FUNCTION_BLOCK PUBLIC FB_CNC EXTENDS FB_EventLogger
VAR_INPUT
	CalibrationCam						: ARRAY[0..HLI_SYS_AX_MAXIDX] OF BOOL;
	LogAxisNo							: ARRAY[0..HLI_SYS_AX_MAXIDX] OF INT;// EtherCAT ID of Axis
	MaxChannelIdx						: INT := 0;	//Max index of channel that is used starting at 0, example: 1 -> totally 2 channels, maximum of 11 (12 channels) is allowed here *)
	Energize							: BOOL;// CNC Energised Flag
END_VAR
VAR_OUTPUT
	
END_VAR
VAR_IN_OUT	                			
	Control								: ST_System;
	Spindle								: ST_Spindle;						//Spindle interface	
END_VAR    
VAR 
	_AxisTorqueLimit					AT %Q* : ARRAY [0..4] OF UINT;								//Bipolar Torque Limit for axes (mapped from drive)
	_DrivePowerManagementStatusWords AT %I* :ARRAY [0..4] OF INT;									//Power management status to detect drives dropping power to ensure rehoming occurs.
	
	_Axis								: ARRAY[0..HLI_SYS_AX_MAXIDX] OF FB_CNCAxis;	//Axis data struct
	{attribute 'tc_no_symbol'}
	_Channel							: ARRAY[0..3] OF HLI3_CNCChannel;	//Channel data struct
	_MachineMode						: ARRAY[0..3] OF ST_MachineMode;	//Machine mode data struct
	_ManualMode							: ST_Selection;						//Manual Mode Selection
	_AutomaticMode						: ST_Selection;						//Automatic Mode Selection
	_MDIMode							: ST_Selection;						//MDI Mode Selection
	_HandwheelMode						: ST_Selection;						//Handwheel Mode Selection
	_StandbyMode						: ST_Selection;						//Standby Mode Selection
	_ReferenceMode						: ST_Selection;						//Reference Mode Selection
	_ManHome							: ST_Selection;						//Manual Home Selection
	_RetractTool						: ST_Selection;						//Retract tool from workpiece
	_SpindleWarmup						: ST_Selection;						//Warm up Spindle
	_AxisNames							: ARRAY[0..4] OF STRING;			//Individual Axis Names for HMI
	_AxisInManual						: ARRAY[0..4] OF BOOL;				//Axis in Manual Flag
	_SelectedChannel					: INT := 0;
	_SelectedAxis						: INT := 0;							//Axis Index Selected from HMI
	_SpindleVelocity					: UINT;								//Spindle Velocity Status
	_SpindleRev							: DINT;								//Spindle Revolution Command
	_AutoEn								: BOOL;								//Auto Enable
	_AutoHome							: BOOL;								//Command Home Drive Auto
	_AxisEnabled						: BOOL;								//All Axes are enabled
	_ManualModeJog						: BOOL;								//Manual Jog Mode
	_ManualModeInc						: BOOL;								//Manual Increment Mode
	_FeedOverride						: UINT := 100;
	_Fault								: BOOL;	     						//Device Fault
	_FaultTimer_ET						: REAL;								//Fault timer elapsed
	_Alarm								: BOOL;								//Device Alarm         
	_Warning							: BOOL;								//Device Warning   
	{attribute 'tc_no_symbol'}
	_ParkMDIString						: STRING;							//Parking MDI String   
	{attribute 'tc_no_symbol'}  
	_AlarmNum							: UDINT;							//Device Alarm Number  
	{attribute 'tc_no_symbol'}
	_WarningNum							: DINT;								//Device Warning Number
	{attribute 'tc_no_symbol'}
	_R_Trig								: ARRAY[0..19] OF R_TRIG;			//Private Rising Edge Triggers
	_HandwheelAxisIsSelected			: BOOL;								//True when axis selected on handwheel
	_Handwheel 							: ST_Handwheel; 					//Handwheel controller inputs
	_ProgramEnd							: ARRAY[0..3] OF BOOL;				//Program End
	_CurrentLine						: DINT;								//N function of currently running program (i.e. N60 -> 60)
	_CurrentNCProgram					: STRING;							//Program currently running in CNC kernal
	_NCProgramCode						: STRING(15000);					//Code of program for reloading into HMI text display\
END_VAR
VAR PERSISTENT                      	
	_Name								: STRING[15];						//Name for HMI
	_Description						: STRING[40];						//Description for HMI
	_AlarmMute							: BOOL;								//Alarm Mute
	_FaultTimer_PT						: REAL;								//Fault timer preset time	
	_Homed								: BOOL;								//Servo is Homed
	_Variables							: ARRAY [0..9] OF ST_Variable;				//Device Associated Varibles Array	
	_ToolData							: ARRAY [0..6] OF ST_CNC_TOOL_DATA_EXT;		//Data for tools
	_PositionOffset						: ARRAY[0..HLI_SYS_AX_MAXIDX] OF LREAL;		//Home position offsets for Axes
	_ParkPositions						: ARRAY[0..HLI_SYS_AX_MAXIDX] OF INT;		//Park positions for Axes
	_pVE_Chan0							: POINTER TO ST_VE_CHAN0;					//Channel 0 User defined Variables
	_Referencing						: E_CNC_HomingMethod; 						//Method to home
	_MeasurementOrder					: ARRAY[0..5] OF UINT :=[2,3,4,1,0];		//Measurement Axis Index Order i.e [2,3,4,1,0] Would be the same as G74 X5 Y4 Z1 C3 A2
	_MeasurementMDIString				: ARRAY[0..5] OF STRING := ['G100 X-10000$R$NM50$R$NM53$R$NG4 1$R$NM51$R$N#PUT AX [X] $R$NM52$R$N#CALL AX [X,11,0]$R$NM54$R$N',
																	'G100 Y-10000$R$NM50$R$NM53$R$NG4 1$R$NM51$R$N#PUT AX [Y] $R$NM52$R$N#CALL AX [Y,10,1]$R$NM54$R$N',
																	'G100 Z1000$R$NM50$R$NM53$R$NG4 1$R$NM51$R$N#PUT AX [Z] $R$NM52$R$N#CALL AX [Z,7,2]$R$NM54$R$N',
																	'G100 C-1000$R$NM50$R$NM53$R$NG4 1$R$NM51$R$N#PUT AX [C] $R$NM52$R$N#CALL AX [C,8,3]$R$NM54$R$N',
																	'G100 A1000$R$NM50$R$NM53$R$NG4 1$R$NM51$R$N#PUT AX [A] $R$NM52$R$N#CALL AX [A,9,4]$R$NM54$R$N',
																	''];//Measurement MDI String

END_VAR

HLI3_Init(); 
M_WarningMonitor();
M_AlarmMonitor();

(* Call CNC related code only if the HLI has been initialized succesfully! *)
IF CNCSystem.bHLIInit THEN
	M_AxesHandler();    	
	M_ManualMode(_Chan:= _SelectedChannel);
	M_ChannelHandler();	
	M_VariableViewer();	
	M_Selections(_Chan:= _SelectedChannel);	
	M_Spindle(_Chan:= _SelectedChannel);
	M_ToolHandler(_Chan:= _SelectedChannel);
	M_Homing(_Chan:= _SelectedChannel);

  //Mod from Local
  //Mod on local pre pull
END_IF

{attribute 'monitoring' := 'variable'}
PROPERTY PUBLIC Alarm : Bool
GET
Alarm := _Alarm;
END_GET
END_PROPERTY

{attribute 'monitoring' := 'variable'}
PROPERTY PUBLIC AlarmMute : BOOL
SET
AlarmMute := _AlarmMute;
END_SET
END_PROPERTY

{attribute 'monitoring' := 'variable'}
PROPERTY PUBLIC AutoHome : Bool
SET
_AutoHome := AutoHome;
END_SET
END_PROPERTY

{attribute 'monitoring' := 'variable'}
PROPERTY PUBLIC AxisEnabled : Bool
GET
AxisEnabled := _AxisEnabled;
END_GET
END_PROPERTY

{attribute 'monitoring' := 'variable'}
PROPERTY PUBLIC Description : String[40]
GET
Description := _Description;
END_GET
SET
_Description := Description;
END_SET
END_PROPERTY

{attribute 'monitoring' := 'variable'}
PROPERTY PUBLIC Fault : Bool
SET
_Fault := Fault;
END_SET
END_PROPERTY

{attribute 'monitoring' := 'variable'}
PROPERTY PUBLIC FaultTimer_ET : real
GET
FaultTimer_ET := _FaultTimer_ET;
END_GET
END_PROPERTY

{attribute 'monitoring' := 'variable'}
PROPERTY PUBLIC FaultTimer_PT : real
GET
FaultTimer_PT := _FaultTimer_PT;
END_GET
SET
_FaultTimer_PT := FaultTimer_PT;
END_SET
END_PROPERTY

PROPERTY PUBLIC FeedOverride : UINT
GET
FeedOverride:= _FeedOverride;
END_GET
SET
_FeedOverride:= FeedOverride;
END_SET
END_PROPERTY

PROPERTY PUBLIC HandwheelSelected : BOOL
GET
HandwheelSelected:= (_MachineMode[0].ManualMode.nManualTyp = 1);
END_GET
END_PROPERTY

{attribute 'monitoring' := 'variable'}
PROPERTY PUBLIC Homed : Bool
GET
Homed := _Homed;
END_GET
END_PROPERTY

METHOD PRIVATE M_AlarmMonitor
VAR_INPUT
END_VAR
VAR_INST // added by the converter: edge detectors and wires of the graphical bodies
    _w1, _w2, _w3, _w4, _w5 : BOOL;
    _rt1 : R_TRIG;
END_VAR
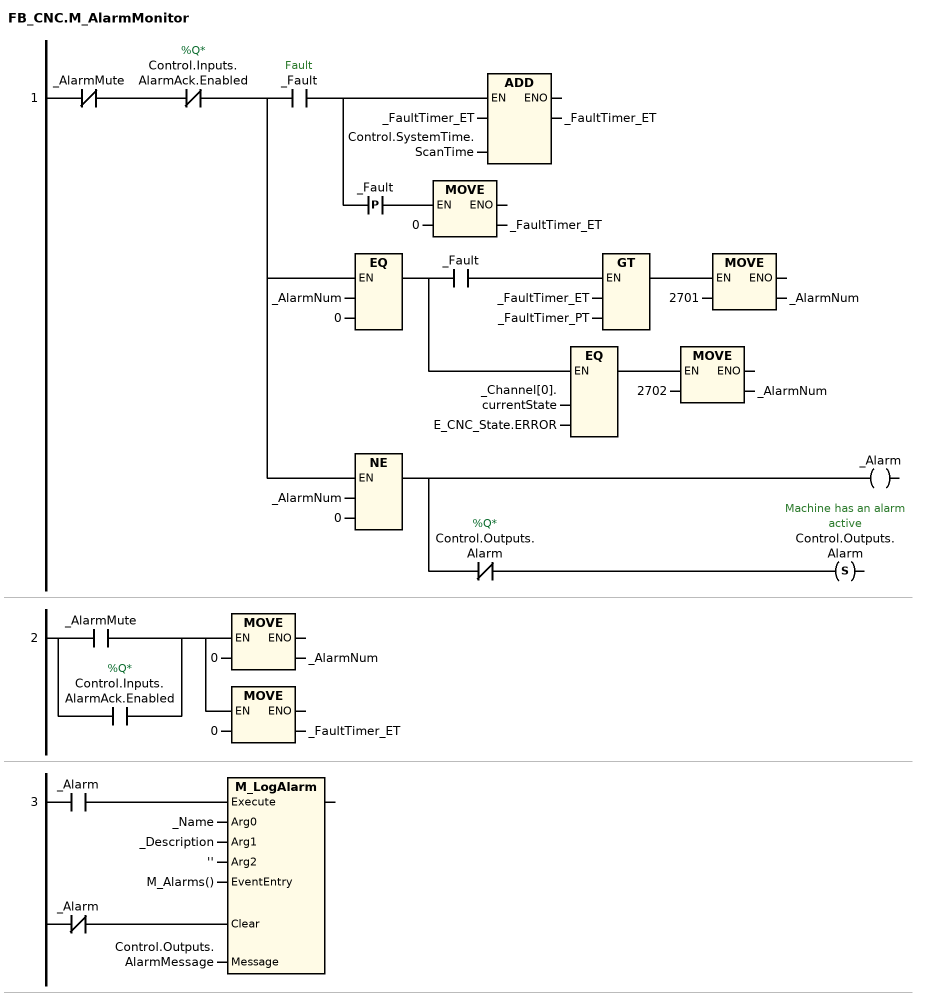
// NETWORK 1
//   Control.Inputs.AlarmAck.Enabled: AT %Q*
//   _Fault: Fault
//   _FaultTimer_ET: Fault timer elapsed
//   Control.SystemTime.ScanTime: Last scan time (Seconds)
//   _FaultTimer_PT: Fault timer preset time
//   Control.Outputs.Alarm: AT %Q* | Machine has an alarm active
_w1 := NOT _AlarmMute AND NOT Control.Inputs.AlarmAck.Enabled;
_w2 := _w1 AND _Fault;
IF _w2 THEN _FaultTimer_ET := _FaultTimer_ET + Control.SystemTime.ScanTime; END_IF
_rt1(CLK := _Fault);
IF _w2 AND _rt1.Q THEN _FaultTimer_ET := 0; END_IF
_w3 := _w1 AND _AlarmNum = 0;
IF _w3 AND _Fault AND _FaultTimer_ET > _FaultTimer_PT THEN _AlarmNum := 2701; END_IF
IF _w3 AND _Channel[0].currentState = E_CNC_State.ERROR THEN _AlarmNum := 2702; END_IF
_w4 := _w1 AND _AlarmNum <> 0;
_Alarm := _w4;
Control.Outputs.Alarm S= _w4 AND NOT Control.Outputs.Alarm;

// NETWORK 2
//   Control.Inputs.AlarmAck.Enabled: AT %Q*
//   _FaultTimer_ET: Fault timer elapsed
_w5 := _AlarmMute OR Control.Inputs.AlarmAck.Enabled;
IF _w5 THEN _AlarmNum := 0; END_IF
IF _w5 THEN _FaultTimer_ET := 0; END_IF

// NETWORK 3
M_LogAlarm(Execute := _Alarm, Arg0 := _Name, Arg1 := _Description, Arg2 := '', EventEntry := M_Alarms(), Clear := NOT _Alarm, Message := Control.Outputs.AlarmMessage);
END_METHOD

METHOD PRIVATE M_Alarms : TcEventEntry
VAR_INPUT
END_VAR
CASE _AlarmNum OF
	2701: M_Alarms:= TC_Events.TcCnc.A_2701;//Alarm	
	2702: M_Alarms:= TC_Events.TcCnc.A_2702;//Mode Error					
ELSE
	M_Alarms:= TC_Events.TcCnc.A_Undefined;
END_CASE
END_METHOD

METHOD PRIVATE M_AxesHandler
VAR_INST
	{attribute 'tc_no_symbol'}
	_HliAxisIdx					: INT;				//Loop index	
	{attribute 'tc_no_symbol'}			
	_FirstSpindle				: INT := -1;		//Spindle HLI index
	{attribute 'tc_no_symbol'}
	_fbAxesError 				: FB_AxesError;		//Axes error
END_VAR
_fbAxesError(bReset := (_Alarm AND Control.Inputs.AlarmAck.Enabled));
_AxisEnabled := TRUE;   
FOR _HliAxisIdx := 0 TO UDINT_TO_INT(gNrAx-1) DO			
	_Axis[_HliAxisIdx](bCalibrationCam:= CalibrationCam[_HliAxisIdx],
		bEnable	:= _AutoEn,
		nLogAxisNo := LogAxisNo[_HliAxisIdx]);
	_Axis[_HliAxisIdx].stOptions.bProbingSignal:= CalibrationCam[_HliAxisIdx];
		
	IF _HliAxisIdx <= UDINT_TO_INT(gNrAx-2) THEN
		_AxisNames[_HliAxisIdx] := gpCh[0]^.bahn_state.coord_r[_HliAxisIdx].axis_name_r.zeichen;
		_AxisInManual[_HliAxisIdx] := _MachineMode[0].ManualMode.nLogAxisNumber = INT_TO_UINT(_Axis[_HliAxisIdx].nLogAxisNo);
		_Axis[_HliAxisIdx].stOptions.bProbingSignal := CalibrationCam[_HliAxisIdx];	
		IF (NOT _Axis[_HliAxisIdx].stStatus.bIsEnabled) THEN    // if one axis status is "not enabled" -> reset PLCStatusAxisEnabled
			_AxisEnabled := FALSE;
		END_IF
	END_IF
		
		IF HLI3_CheckAxisValid(_HliAxisIdx) THEN
			IF _FirstSpindle = -1 AND gpAx[_HliAxisIdx]^.ipo_state.spindle_axis_r THEN  (* store HLIIndex of first spindle *)
				_FirstSpindle := _HliAxisIdx;
			END_IF
		END_IF
		
END_FOR
END_METHOD

METHOD M_ChannelHandler
VAR_INST
	{attribute 'tc_no_symbol'}
	_Chan					: INT;								//Channel index
	{attribute 'tc_no_symbol'}
	_OldSelectedChannel		: UDINT;							//Previous channel index
	{attribute 'tc_no_symbol'}
	_stOptions				: ST_CNC_CH_Options;				//HLI options for structure 
	{attribute 'tc_no_symbol'}
	_ChannelSignals			: ST_ChannelSignals;				//HLI channel signal structure
	{attribute 'tc_no_symbol'}
	_BlockSearch			: ARRAY[0..3] OF HLI3_BlockSearch;	//HLI block search structure
	{attribute 'tc_no_symbol'}
	_ErrorHandler			: ARRAY[0..3] OF FB_ChannelError;	//HLI channel error structure				
END_VAR
IF (_OldSelectedChannel <>INT_TO_UDINT(_SelectedChannel)) THEN
	_ChannelSignals.SingleBlock 		:= _MachineMode[_SelectedChannel].ChannelSignals.SingleBlock;
	_ChannelSignals.PrgBlockIgnore		:= _MachineMode[_SelectedChannel].ChannelSignals.PrgBlockIgnore;
	_ChannelSignals.M01Stop 			:= _MachineMode[_SelectedChannel].ChannelSignals.M01Stop;
	_ChannelSignals.Backward 			:= _MachineMode[_SelectedChannel].ChannelSignals.Backward;
	_ChannelSignals.FeedHold 			:= _MachineMode[_SelectedChannel].ChannelSignals.FeedHold;
	_OldSelectedChannel 				:= INT_TO_UDINT(_SelectedChannel);
END_IF

_MachineMode[_SelectedChannel].ChannelSignals.SingleBlock 	:= _ChannelSignals.SingleBlock;
_MachineMode[_SelectedChannel].ChannelSignals.PrgBlockIgnore:= _ChannelSignals.PrgBlockIgnore;
_MachineMode[_SelectedChannel].ChannelSignals.M01Stop 		:= _ChannelSignals.M01Stop;
_MachineMode[_SelectedChannel].ChannelSignals.Backward 		:= _ChannelSignals.Backward;
_MachineMode[_SelectedChannel].ChannelSignals.FeedHold 		:= _ChannelSignals.FeedHold;

_stOptions.bReferenceModeStartRequired := FALSE;
//_stOptions.bDisableCNCPLCWatchDog := TRUE;

FOR _Chan := 0 TO MaxChannelIdx DO
	IF (HLI3_CheckChannelValid(_Chan)) THEN		
		
		_MachineMode[_Chan].Mode 	:= _Channel[_Chan].currentMode;
		_MachineMode[_Chan].State	:= _Channel[_Chan].currentState;
		_ErrorHandler[_Chan](nChanIdx	:= _Chan);				

		_Channel[_Chan]
			(nChanIdx			:= _Chan,							
			 bModeStandby		:= _MachineMode[_Chan].Standby,
			 bModeAutomatic		:= _MachineMode[_Chan].Automatic,
			 bModeManual		:= _MachineMode[_Chan].Manual,
			 bModeMDI			:= _MachineMode[_Chan].MDI,	 
			 bModeReference		:= _MachineMode[_Chan].Homing,
			 bStateSelect		:= _MachineMode[_Chan].Select,
			 bStateReady		:= _MachineMode[_Chan].Ready,
			 bStateStart		:= _MachineMode[_Chan].Start,
			 bStateStop			:= _MachineMode[_Chan].Stop,
			 bStateReset		:= _MachineMode[_Chan].Reset,
			 nFeedOverride		:= _FeedOverride * 10,
			 nRapidFeedOverride := _FeedOverride * 10, 
			 sProgramName		:= _MachineMode[_Chan].ProgramName,			 
			 sMDIString			:= _MachineMode[_Chan].MDIString,
			 bBackwardMotion	:= _MachineMode[_Chan].ChannelSignals.Backward,
			 bPrgBlockIgnore	:= _MachineMode[_Chan].ChannelSignals.PrgBlockIgnore,
			 bFeedHold			:= _MachineMode[_Chan].ChannelSignals.FeedHold,
			 bSingleBlock		:= _MachineMode[_Chan].ChannelSignals.SingleBlock,
			 bDoSingleBlock		:= _MachineMode[_Chan].ChannelSignals.DoSingleBlock,
			 bM01Stop			:= _MachineMode[_Chan].ChannelSignals.M01Stop,
			 nSyntaxCheck		:= _MachineMode[_Chan].SyntaxCheck.nType,
			 bM30Acknowledgement:= TRUE,
			 stManualModeParameter  	 	 := stManualModeParameter[_Chan],
			 stManualModeControlElements	 := stManualModeControlElements[_Chan],
			 stManualModeControlElementState := stManualModeControlElementState,
			 stOptions			:= 	_stOptions
			);
			
		_r_trig[_Chan](CLK:= gpCh[_Chan]^.bahn_state.program_end_r);
		_ProgramEnd[_Chan]:= _r_trig[_Chan].Q;
		
		_BlockSearch[_Chan]
			(nChanIdx			:= _Chan,
			 bStartRead      	:= _MachineMode[_Chan].BlockSearch.bStartRead,   (* Edge signal *)
			 bStartWrite     	:= _MachineMode[_Chan].BlockSearch.bStartWrite,  (* Edge signal *)
			 BlockSearch		:= _MachineMode[_Chan].BlockSearch
			);
		
		CNCSystem.Channel[_Chan].ActDistance 	:= DINT_TO_LREAL(_BlockSearch[_Chan].coveredDistance_AfterReset) / 10.0;
		CNCSystem.Channel[_Chan].ActBlockCount 	:= _BlockSearch[_Chan].actualBlockCount_AfterReset;
						
	END_IF
END_FOR

_CurrentNCProgram := gpCh[0]^.bahn_state.file_name_r.zeichen;
_CurrentLine:= gpCh[0]^.bahn_state.block_nr_r;
END_METHOD

METHOD PRIVATE M_Homing
VAR_INPUT
	{attribute 'tc_no_symbol'}
	_Chan								 : INT;									//Channel index
END_VAR
VAR_INST
	{attribute 'tc_no_symbol'}
	_Step                  			 	 : ARRAY[0..3] OF INT;					//Step counter
	{attribute 'tc_no_symbol'}
	_Axe					 			 : UINT;								//Axes index
	{attribute 'tc_no_symbol'}
	_SetDrivePosition					 : BOOL;								//Set drive position
	{attribute 'tc_no_symbol'}
	_DeleteDrivePosition				 : BOOL;								//Delete drive position
	{attribute 'tc_no_symbol'}	
	_fb_CNCAX5000SetPositionOffset		 : FB_CNCAX5000SetPositionOffset;		//Sets encoder position in drive memory
	{attribute 'tc_no_symbol'}
	_fb_CNCAX5000DeletePositionOffset	 : FB_CNCAX5000DeletePositionOffset;	//Clears drive memory
END_VAR
IF _MachineMode[_Chan].State = E_CNC_State.ERROR OR Control.PackMLState.Stopped THEN
   _Step[_Chan] := 0;
END_IF
 
CASE _Referencing OF

//Homing Method with Calibration Cam. This method uses the Position Offsets stored in the CNC Params. The encoder position is NOT stored in memory.
E_CNC_HomingMethod.Homing:

	CASE _Step[_Chan] OF
		0: //Idle
			IF _AutoHome AND NOT _Alarm THEN
				_Homed := FALSE;
				_Axe:=0;
			    _Step[_Chan] := 1;
			ELSIF _ManHome.Queued AND NOT _Alarm THEN
				_Homed := FALSE;
				IF _ManHome.Enabled THEN
					_Axe:=INT_TO_UINT(_SelectedAxis);
					_Step[_Chan] := 10;
				END_IF
			END_IF
		
		1://Update Homing Offsets
			_Axis[0].fRefOffset:= _PositionOffset[0];
			_Axis[0].bSetRefOffset:= TRUE;
			_Axis[1].fRefOffset:= _PositionOffset[1];
			_Axis[1].bSetRefOffset:= TRUE;
			_Axis[2].fRefOffset:= _PositionOffset[2];
			_Axis[2].bSetRefOffset:= TRUE;
			_Axis[3].fRefOffset:= _PositionOffset[3];
			_Axis[3].bSetRefOffset:= TRUE;
			_Axis[4].fRefOffset:= _PositionOffset[4];
			_Axis[4].bSetRefOffset:= TRUE;

			_Step[_Chan] := 2;
	
	
		2://Enable Homing
			_MachineMode[0].Homing:= TRUE;

			IF _Axis[0].stStatus.bHomingDone AND _Axis[1].stStatus.bHomingDone AND 
				_Axis[2].stStatus.bHomingDone AND _Axis[3].stStatus.bHomingDone AND _Axis[4].stStatus.bHomingDone THEN
					_Step[_Chan] := 3;
			END_IF
	
		3: //Wait for CNC to reach park positions
		 	IF _MachineMode[_Chan].State = E_CNC_State.READY THEN
		     	_Step[_Chan] := 4;
		 	END_IF
		
		4://Set mode to standby	
			_Homed := TRUE;
			_MachineMode[_Chan].Standby := TRUE;
			IF NOT _Autohome AND NOT _ManHome.Enabled AND _MachineMode[_Chan].Mode = E_CNC_Mode.STANDBY_MODE THEN
				_Step[_Chan] := 0;
			END_IF
			
		//Single Axis Manual Home
		10://Set MDI Mode
			_MachineMode[_Chan].MDI := TRUE;
			IF _MachineMode[_Chan].Mode = E_CNC_Mode.MDI_MODE THEN
				_Step[_Chan] := 11;
	    	END_IF
			
		11://Set homing string for indiviudal axis
			CASE _Axe OF
				0: _MachineMode[_Chan].MDIString := 'G74 X0';
				1: _MachineMode[_Chan].MDIString := 'G74 Y0';
				2: _MachineMode[_Chan].MDIString := 'G74 Z0';
				3: _MachineMode[_Chan].MDIString := 'G74 C0';
				4: _MachineMode[_Chan].MDIString := 'G74 A0';
			END_CASE
			_MachineMode[_Chan].Start := TRUE;
			_SetDrivePosition := FALSE;
	 		_Step[_Chan] := 12;
			
		12://Wait for CNC ready state
			IF _MachineMode[_Chan].State = E_CNC_State.READY THEN
	       		_Step[_Chan] := 13;
	    	END_IF
			
		13://Park Axis
			_MachineMode[_Chan].MDIString := CONCAT(_AxisNames[_SelectedAxis],TO_STRING(_ParkPositions[_SelectedAxis]));
			_MachineMode[_Chan].Start := TRUE;
			_Step[_Chan] := 14;
		
		14: //Wait for CNC to start moving to park positions
		 	IF _MachineMode[_Chan].State = E_CNC_State.ACTIVE THEN
		     	_Step[_Chan] := 15;
		 	END_IF		
			
		15: //Wait for CNC to reach park positions
		 	IF _MachineMode[_Chan].State = E_CNC_State.READY THEN
		     	_Step[_Chan] := 16;
		 	END_IF
		
		16://Set mode to standby	
			_Homed := TRUE;
			_MachineMode[_Chan].Standby := TRUE;
			IF NOT _Autohome AND NOT _ManHome.Enabled AND _MachineMode[_Chan].Mode = E_CNC_Mode.STANDBY_MODE THEN
				_Step[_Chan] := 0;
			END_IF
	END_CASE		


//Measurement Method With Probing Signal. This method uses the Position Offsets stored in the PLC. The encoder position IS stored in memory.
E_CNC_HomingMethod.Measurment:

	CASE _Step[_Chan] OF
		0: //Idle
			IF _AutoHome AND NOT _Alarm THEN
				_SetDrivePosition := FALSE;
				FOR _Axe := 0 TO UDINT_TO_UINT(gNrAx-2) DO
					_Axis[_MeasurementOrder[_Axe]].bSetRefOffset := FALSE;
					_Axis[_MeasurementOrder[_Axe]].stOptions.bResetCalibration := TRUE;
				END_FOR;
				_Homed := FALSE;
				_Axe:= 0;
			    _Step[_Chan] := 1;
			ELSIF _ManHome.Queued AND NOT _Alarm THEN
				_Homed := FALSE;
				IF _ManHome.Enabled THEN
					_Axe:=INT_TO_UINT(_SelectedAxis);
					_Step[_Chan] := 1;
				END_IF
			END_IF
			
		1://Enable Axes and set Standby Mode
			_AutoEn := TRUE;
			_MachineMode[_Chan].Standby := TRUE;
			IF _AxisEnabled AND _MachineMode[_Chan].Mode = E_CNC_Mode.STANDBY_MODE THEN
				_Step[_Chan] := 2;
			END_IF
	    	
	    2: //Set MDI mode
			_MachineMode[_Chan].MDI := TRUE;
			IF _MachineMode[_Chan].Mode = E_CNC_Mode.MDI_MODE THEN
				_Step[_Chan] := 3;
	    	END_IF
			
		3: //Reset homing done bool to allow ignorance of software limits
			IF _Axis[_MeasurementOrder[_Axe]].stStatus.bHomingDone = FALSE THEN
				_Axis[_MeasurementOrder[_Axe]].stOptions.bResetCalibration := FALSE;	
				_Step[_Chan] := 4;
			END_IF
			
	    4: //Create homing MDI string
			IF _ManHome.Enabled THEN
				_MachineMode[_Chan].MDIString := _MeasurementMDIString[_Axe];
			ELSE
				_MachineMode[_Chan].MDIString := _MeasurementMDIString[_MeasurementOrder[_Axe]];	
			END_IF
			_MachineMode[_Chan].Start := TRUE;
			_SetDrivePosition := FALSE;
	 		_Step[_Chan] := 5;
		
	    5: //Wait for CNC to start moving to home positions
	    	IF _MachineMode[_Chan].State = E_CNC_State.ACTIVE THEN
	       		_Step[_Chan] := 6;
	    	END_IF	
	
		6://Wait for CNC to reach home positions
		
				//M50 Clear Reference Flag
				IF CNCSystem.Channel[0].M[50].bState_rw THEN
					_Axis[_MeasurementOrder[_Axe]].stOptions.bResetCalibration := TRUE;
					IF _Axis[_MeasurementOrder[_Axe]].stStatus.bHomingDone = FALSE THEN
						_Axis[_MeasurementOrder[_Axe]].stOptions.bResetCalibration := FALSE;
						CNCSystem.Channel[0].M[50].bState_rw := FALSE;
					END_IF
				END_IF
				
				//M51 Set Drive Position
				IF CNCSystem.Channel[0].M[51].bState_rw THEN
					_SetDrivePosition := TRUE;
				END_IF
				IF _Axis[_MeasurementOrder[_Axe]].stStatus.fActPosACS > (_PositionOffset[_MeasurementOrder[_Axe]] -1) AND  _Axis[_MeasurementOrder[_Axe]].stStatus.fActPosACS < (_PositionOffset[_MeasurementOrder[_Axe]] +1) THEN
					CNCSystem.Channel[0].M[51].bState_rw := FALSE;
					_SetDrivePosition := FALSE;
				END_IF 
				
				//M52 Set Axis as Homed
				IF CNCSystem.Channel[0].M[52].bState_rw THEN
					_Axis[_MeasurementOrder[_Axe]].fRefOffset := 0;
					_Axis[_MeasurementOrder[_Axe]].bSetRefOffset := TRUE;
					IF _Axis[_MeasurementOrder[_Axe]].stStatus.bHomingDone = TRUE THEN
						CNCSystem.Channel[0].M[52].bState_rw := FALSE;
						_Axis[_MeasurementOrder[_Axe]].bSetRefOffset := FALSE;
					END_IF
				END_IF
				
				//M53 Disable Axis
				IF CNCSystem.Channel[0].M[53].bState_rw THEN
					_AutoEn := FALSE;
					IF NOT _Axis[_MeasurementOrder[_Axe]].stStatus.bIsEnabled THEN
						CNCSystem.Channel[0].M[53].bState_rw := FALSE;
					END_IF
				END_IF
				
				//M54 Enable Axis
				IF CNCSystem.Channel[0].M[54].bState_rw THEN
					_AutoEn := TRUE;
					IF _Axis[_MeasurementOrder[_Axe]].stStatus.bIsEnabled THEN
						CNCSystem.Channel[0].M[54].bState_rw := FALSE;
						_Step[_Chan] := 7;	
					END_IF
				END_IF
				
	    7: //Wait for CNC to be Ready
	    	IF _MachineMode[_Chan].State = E_CNC_State.READY THEN
	       		IF (_ManHome.Enabled OR _Axe >= (gNrAx-3)) THEN//)>= 1 THEN
					_Step[_Chan] := 8;
				ELSE
					_Axe:=_Axe+1;
					_Step[_Chan] := 3;
				END_IF
	    	END_IF	
				
		8://Create parking MDI string
			IF _ManHome.Enabled THEN
				_ParkMDIString := CONCAT(_AxisNames[_SelectedAxis],TO_STRING(_ParkPositions[_SelectedAxis]));
			ELSE	
				FOR _Axe := 0 TO UDINT_TO_UINT(gNrAx-2) BY 1 DO	
					IF _Axe = 0 THEN
						_ParkMDIString	:= concat(_AxisNames[_Axe],TO_STRING(_ParkPositions[_Axe]));
					ELSE
						_ParkMDIString	:= concat(_ParkMDIString,concat(' ', concat(_AxisNames[_Axe],TO_STRING(_ParkPositions[_Axe]))));
					END_IF
				END_FOR	
			END_IF
			_MachineMode[_Chan].MDIString := _ParkMDIString;
			_MachineMode[_Chan].Start := TRUE;
			_Step[_Chan] := 9;
		
		9: //Wait for CNC to start moving to park positions
		 	IF _MachineMode[_Chan].State = E_CNC_State.ACTIVE THEN
		     	_Step[_Chan] := 10;
		 	END_IF		
			
		10: //Wait for CNC to reach park positions
		 	IF _MachineMode[_Chan].State = E_CNC_State.READY THEN
		     	_Step[_Chan] := 11;
		 	END_IF
		
		11://Set mode to standby	
			_Homed := TRUE;
			_MachineMode[_Chan].Standby := TRUE;
			IF NOT _Autohome AND NOT _ManHome.Enabled AND _MachineMode[_Chan].Mode = E_CNC_Mode.STANDBY_MODE THEN
				_Step[_Chan] := 0;
			END_IF
			
	END_CASE

END_CASE

//Delete Position Offset
_fb_CNCAX5000DeletePositionOffset(nLogAxisNo:= TO_UINT(_Axis[_MeasurementOrder[_Axe]].nLogAxisNo), Execute:= _DeleteDrivePosition, Memory:= tc3_cnc_drive.E_PositionOffsetMemory.ePositionOffsetMemory_Drive);

//Set Position Offset
_fb_CNCAX5000SetPositionOffset(nLogAxisNo:= TO_UINT(_Axis[_MeasurementOrder[_Axe]].nLogAxisNo), Execute:= _SetDrivePosition, Position:= _PositionOffset[_MeasurementOrder[_Axe]], Memory:= tc3_cnc_drive.E_PositionOffsetMemory.ePositionOffsetMemory_Drive);
END_METHOD

METHOD PRIVATE M_ManualMode
VAR_INPUT
	{attribute 'tc_no_symbol'}
	_Chan								 : INT;									//Channel index
END_VAR	
VAR_INST
	{attribute 'tc_no_symbol'}
	_fbUintUdInt						 : ARRAY [0..3] OF FB_Uint_Udint;		//Uint to udint FB
	{attribute 'tc_no_symbol'}
	_HandWheelBig						 : UDINT;								//Handwheel value
END_VAR
IF (HLI3_CheckChannelValid(_Chan)) THEN

	stManualModeParameter[_Chan].stChannelParameter.nChanIdx := _Chan;       (* Channel 1 *)
	stManualModeParameter[_Chan].stChannelParameter.nInc := _MachineMode[_Chan].ManualMode.nInc * 10;
	stManualModeParameter[_Chan].stChannelParameter.bG200ConfigurationViaPLC := TRUE;		
	
	stManualModeParameter[_Chan].stChannelParameter.eManualType := UINT_TO_INT(_MachineMode[_Chan].ManualMode.nManualTyp);			
	IF (stManualModeParameter[_Chan].stChannelParameter.eManualType = E_CNC_ManualType.Handwheel AND _Chan <> _SelectedChannel) THEN	(* if in Handwheel mode and the channel is NOT selected -> leave handwheel mode and change to TippMode*)
		stManualModeParameter[_Chan].stChannelParameter.eManualType := E_CNC_ManualType.TippMode;
	END_IF		
	
	stManualModeParameter[_Chan].stChannelParameter.stManualOption.bTrafoActive := _MachineMode[_Chan].ManualMode.stManualOption.bTrafoActive;
	stManualModeParameter[_Chan].stChannelParameter.stManualOption.bEcsActive := _MachineMode[_Chan].ManualMode.stManualOption.bEcsActive;
	stManualModeParameter[_Chan].stChannelParameter.stManualOption.eZeroOffset := _MachineMode[_Chan].ManualMode.stManualOption.eZeroOffset;					

	_ManualModeJog:=(_MachineMode[_SelectedChannel].ManualMode.nManualTyp=2) AND _Channel[_SelectedChannel].stCmdModesStates.stModes.Manual;
	_ManualModeInc:=(_MachineMode[_SelectedChannel].ManualMode.nManualTyp=3) AND _Channel[_SelectedChannel].stCmdModesStates.stModes.Manual;
	
	stManualModeParameter[_Chan].stAxisParameter.stControlUnit[0].nLogAxisNr := _MachineMode[_Chan].ManualMode.nLogAxisNumber;   (* Log. Achs Nummer *)
	IF stManualModeParameter[_Chan].stAxisParameter.stControlUnit[0].nLogAxisNr = 0 THEN
		stManualModeParameter[_Chan].stAxisParameter.stControlUnit[0].nLogAxisNr := gpCh[_Chan]^.bahn_state.coord_r[0].log_achs_nr_r;
		_MachineMode[_Chan].ManualMode.nLogAxisNumber := gpCh[_Chan]^.bahn_state.coord_r[0].log_achs_nr_r;
	END_IF
	stManualModeParameter[_Chan].stAxisParameter.stControlUnit[0].nSpeed := LREAL_TO_UDINT(_MachineMode[_Chan].ManualMode.nSpeed * (100000/60));//um/min >> mm/sec
	stManualModeControlElements[_Chan].stControlKeys[0].bKeyNeg := _MachineMode[_Chan].ManualMode.bKeyNeg;
	stManualModeControlElements[_Chan].stControlKeys[0].bKeyPos := _MachineMode[_Chan].ManualMode.bKeyPos;
	stManualModeControlElements[_Chan].stControlKeys[0].bKeyRapid := _MachineMode[_Chan].ManualMode.bKeyRapid;
	
	//Handwheel
	IF _Handwheel.xAxisSelect THEN
		_MachineMode[_Chan].ManualMode.nLogAxisNumber := INT_TO_UINT(_Axis[0].nLogAxisNo);
	ELSIF _Handwheel.yAxisSelect THEN
		_MachineMode[_Chan].ManualMode.nLogAxisNumber := INT_TO_UINT(_Axis[1].nLogAxisNo);
	ELSIF _Handwheel.zAxisSelect THEN
		_MachineMode[_Chan].ManualMode.nLogAxisNumber := INT_TO_UINT(_Axis[2].nLogAxisNo);
	ELSIF _Handwheel.aAxisSelect THEN
		_MachineMode[_Chan].ManualMode.nLogAxisNumber := INT_TO_UINT(_Axis[3].nLogAxisNo);
	ELSIF _Handwheel.cAxisSelect THEN
		_MachineMode[_Chan].ManualMode.nLogAxisNumber := INT_TO_UINT(_Axis[4].nLogAxisNo);
	ELSIF _MachineMode[_Chan].ManualMode.nManualTyp = 1 THEN
		_MachineMode[_Chan].ManualMode.nManualTyp := 0;			
	END_IF
	
	IF _Handwheel.x10Resolution THEN
		_MachineMode[_Chan].ManualMode.nHwResolution := 10;
	ELSIF _Handwheel.x100Resolution THEN
		_MachineMode[_Chan].ManualMode.nHwResolution := 100;
	ELSE
		_MachineMode[_Chan].ManualMode.nHwResolution := 1;
	END_IF
		
	stManualModeParameter[_Chan].stChannelParameter.nHandwheelResolution := UDINT_TO_DINT(_MachineMode[_Chan].ManualMode.nHwResolution)* LREAL_TO_DINT(10000);
	_fbUintUdint[_Chan](ninSmall := _Handwheel.Handwheel, nBig := _HandWheelBig);
	stManualModeControlElements[_Chan].nHandwheelinc[0] :=  UDINT_TO_DINT(_HandWheelBig);
	IF _HandWheelBig > 214748364 OR _HandWheelBig = 0 THEN
		_MachineMode[_Chan].ManualMode.nLogAxisNumber := 0;
		_HandWheelBig := 107374182;
	END_IF
END_IF
END_METHOD

METHOD PRIVATE M_Selections
VAR_INPUT
	{attribute 'tc_no_symbol'}
	_Chan					 : INT;
END_VAR
VAR_INST
END_VAR
//Reset
	_MachineMode[_Chan].Reset := Control.Inputs.AlarmAck.Enabled OR Control.Inputs.Reset.Enabled;

//Energize
	_R_Trig[7](CLK:=Energize); 
	IF _R_Trig[7].Q THEN 
		_AutoEn:= TRUE; 
	END_IF
	
	_R_trig[6](CLK:= NOT Energize); 
	IF _R_Trig[6].Q THEN 
		_AutoEn:= FALSE; 
	END_IF

//Stop
	_R_Trig[8](CLK:=Control.PackMLState.Stopping OR Control.PackMLState.Holding);
	_MachineMode[_SelectedChannel].Stop := _R_Trig[8].Q;

//Start
	_R_Trig[9](CLK:= (Control.PackMLState.Starting OR Control.PackMLState.Execute) AND _AxisEnabled);
	_MachineMode[_SelectedChannel].Start := _R_Trig[9].Q;
	
//Standby Mode
	_StandbyMode.Interlock := Control.PackMLState.Execute  OR (_StandbyMode.Enabled AND _MachineMode[_Chan].Mode <> E_CNC_Mode.STANDBY_MODE);
	IF _StandbyMode.Interlock THEN 
		_StandbyMode.Messages := 'CNC Machine Must not be Executing for Standby Mode'; 
	END_IF;
	
	_StandbyMode.Select := (_StandbyMode.Select) AND NOT _StandbyMode.Interlock;
	IF NOT _StandbyMode.Select AND NOT _StandbyMode.Interlock THEN 
		_StandbyMode.Messages := 'CNC Ready for Standby Mode'; 
	END_IF;
	
	_StandbyMode.Queued := _StandbyMode.Select;
	IF _StandbyMode.Queued AND NOT _StandbyMode.Enabled THEN 
		_StandbyMode.Messages := 'CNC Standby Mode Selection Queued'; 
	END_IF;
	
	_R_Trig[10](CLK:= _StandbyMode.Queued); 
	IF _R_Trig[10].Q THEN 
		_MachineMode[_Chan].Standby := TRUE;
	END_IF;
	
	_StandbyMode.Enabled := _StandbyMode.Queued AND _MachineMode[_Chan].Mode = E_CNC_Mode.STANDBY_MODE;
	IF _StandbyMode.Enabled THEN 
		_StandbyMode.Messages := 'CNC Standby Mode Enabled'; 
	END_IF;

//Automatic Mode Selection
	_AutomaticMode.Interlock := Control.PackMLState.Execute AND NOT _AutomaticMode.Enabled OR (_AutomaticMode.Enabled AND _MachineMode[_Chan].Mode <> E_CNC_Mode.AUTOMATIC_MODE);
	IF _AutomaticMode.Interlock THEN 
		_AutomaticMode.Messages := 'CNC Machine Must not be Executing for Automatic Mode Selection'; 
	END_IF;
	
	_AutomaticMode.Select := _AutomaticMode.Select AND NOT _AutomaticMode.Interlock;
	IF NOT _AutomaticMode.Select AND NOT _AutomaticMode.Interlock THEN
 		_AutomaticMode.Messages := 'CNC Ready for Automatic Mode'; 
	END_IF;
	
	_AutomaticMode.Queued := _AutomaticMode.Select;
	IF _AutomaticMode.Queued AND NOT _AutomaticMode.Enabled THEN 
		_AutomaticMode.Messages := 'CNC Automatic Mode Selection Queued'; 
	END_IF;
	
	_R_Trig[11](CLK:= _AutomaticMode.Queued);
	IF _R_Trig[11].Q THEN 
		_MachineMode[_Chan].Automatic := TRUE;
	END_IF;
	
	_AutomaticMode.Enabled := _AutomaticMode.Queued AND _MachineMode[_Chan].Mode = E_CNC_Mode.AUTOMATIC_MODE;
	IF _AutomaticMode.Enabled THEN 
		_AutomaticMode.Messages := 'CNC Automatic Mode Enabled'; 
	END_IF;

//3 MDI Mode Selection
	_MDIMode.Interlock := Control.PackMLState.Execute AND NOT _MDIMode.Enabled  OR (_MDIMode.Enabled AND _MachineMode[_Chan].Mode <> E_CNC_Mode.MDI_MODE);
	IF _MDIMode.Interlock THEN 
		_MDIMode.Messages := 'CNC Machine Must not be Executing for MDI Mode Selection'; 
	END_IF;
	
	_MDIMode.Select := _MDIMode.Select AND NOT _MDIMode.Interlock;
	IF NOT _MDIMode.Select AND NOT _MDIMode.Interlock THEN 
		_MDIMode.Messages := 'CNC Ready for MDI Mode'; 
	END_IF;
	
	_MDIMode.Queued := _MDIMode.Select;
	IF _MDIMode.Queued AND NOT _MDIMode.Enabled THEN 
		_MDIMode.Messages := 'CNC MDI Mode Selection Queued'; 
	END_IF;
	
	_R_Trig[12](CLK:= _MDIMode.Queued); 
	IF _R_Trig[12].Q THEN 
		_MachineMode[_Chan].MDI:= TRUE;
	END_IF;

	_MDIMode.Enabled := _MDIMode.Queued AND _MachineMode[_Chan].Mode = E_CNC_Mode.MDI_MODE;
	IF _MDIMode.Enabled THEN 
		_MDIMode.Messages := 'CNC MDI Mode Enabled'; 
	END_IF;

//Manual Mode Selection
	_ManualMode.Interlock := (NOT control.PackMLState.Stopped AND NOT control.PackMLState.Idle)OR (_ManualMode.Enabled AND ((_MachineMode[_Chan].Mode <> E_CNC_Mode.MANUAL_MODE)OR _R_Trig[15].Q));
	IF _ManualMode.Interlock THEN 
		_ManualMode.Messages := 'CNC Must be in a Stopped or Idle State for Manual Mode'; 
	END_IF;	_R_Trig[13](CLK:= _ManualMode.Queued);
	
	_ManualMode.Select := _ManualMode.Select AND NOT _ManualMode.Interlock;
	IF NOT _ManualMode.Select AND NOT _ManualMode.Interlock THEN 
		_ManualMode.Messages := 'CNC Ready for Manual Mode'; 
	END_IF;
	
	_ManualMode.Queued := _ManualMode.Select;
	IF _ManualMode.Queued AND NOT _ManualMode.Enabled THEN 
		_ManualMode.Messages := 'CNC Manual Mode Selection Queued'; 
	END_IF;

	IF _R_Trig[13].Q THEN 
		_MachineMode[_Chan].ManualMode.nManualTyp := 2;  _MachineMode[_Chan].Manual := TRUE; 
	END_IF;
	
	_ManualMode.Enabled := _ManualMode.Queued AND (_MachineMode[_Chan].ManualMode.nManualTyp<>1) AND _MachineMode[_Chan].Mode = E_CNC_Mode.MANUAL_MODE;
	IF _ManualMode.Enabled THEN 
		_ManualMode.Messages := 'CNC Manual Mode Enabled';
	END_IF;
	
//5 Reference Mode Selection
	_ReferenceMode.Interlock := NOT Control.PackMLState.Resetting OR (_ReferenceMode.Enabled AND _MachineMode[_Chan].Mode <> E_CNC_Mode.REFERENCE_MODE);
	IF _ReferenceMode.Interlock THEN 
		_ReferenceMode.Messages := 'CNC Must be in a Stopped or Resseting State for Reference Mode'; 
	END_IF;
	
	_ReferenceMode.Select := (_ReferenceMode.Select OR _AutoHome OR _ManHome.Enabled) AND NOT _ReferenceMode.Interlock;
	IF NOT _ReferenceMode.Select AND NOT _ReferenceMode.Interlock THEN 
		_ReferenceMode.Messages := 'CNC Ready for Reference Mode'; 
	END_IF;

	_ReferenceMode.Queued := _ReferenceMode.Select;
	IF _ReferenceMode.Queued AND NOT _ReferenceMode.Enabled THEN 
		_ReferenceMode.Messages := 'CNC Reference Mode Selection Queued'; 
	END_IF;

	_ReferenceMode.Enabled := _ReferenceMode.Queued;
	IF _ReferenceMode.Enabled THEN 
		_ReferenceMode.Messages := 'CNC Reference Mode Enabled';
	END_IF;
	
//Handwheel Mode Selected
	_HandwheelMode.Interlock := (NOT control.PackMLState.Stopped AND NOT control.PackMLState.Idle) OR (_HandwheelMode.Enabled AND ((_MachineMode[_Chan].Mode <> E_CNC_Mode.MANUAL_MODE)OR _R_Trig[13].Q));
	IF _HandwheelMode.Interlock THEN 
		_HandwheelMode.Messages := 'CNC Must be in a Stopped or Idle State for Handwheel Mode'; 
	END_IF;

	_HandwheelMode.Select := (_Handwheel.xAxisSelect OR _Handwheel.yAxisSelect OR _Handwheel.zAxisSelect OR _Handwheel.cAxisSelect OR _Handwheel.aAxisSelect) AND NOT _HandwheelMode.Interlock;
	IF NOT _HandwheelMode.Select AND NOT _HandwheelMode.Interlock THEN 
		_HandwheelMode.Messages := 'CNC Ready for Handwheel Mode'; 
	END_IF;

	_HandwheelMode.Queued := _HandwheelMode.Select;
	IF _HandwheelMode.Queued AND NOT _HandwheelMode.Enabled THEN 
		_HandwheelMode.Messages := 'CNC Handwheel Mode Selection Queued'; 
	END_IF;

	_R_Trig[15](CLK:= _HandwheelMode.Queued);
	IF _R_Trig[15].Q THEN 
		_MachineMode[_Chan].ManualMode.nManualTyp := 1; _MachineMode[_Chan].Manual := TRUE; 
	END_IF;

	_HandwheelMode.Enabled := _HandwheelMode.Queued AND (_MachineMode[_Chan].ManualMode.nManualTyp=1) AND _MachineMode[_Chan].Mode = E_CNC_Mode.MANUAL_MODE;
	IF _HandwheelMode.Enabled THEN 
		_HandwheelMode.Messages := 'CNC Handwheel Mode Enabled'; 
	END_IF;

//Manual Home Selection
	_R_Trig[16](CLK:= _Homed);	
	_ManHome.Interlock := (NOT control.PackMLState.Stopped AND NOT control.PackMLState.Resetting) OR _R_Trig[16].Q;
	IF _ManHome.Interlock THEN 
		_ManHome.Messages := 'CNC Must be in a Stopped State for Manual Homing'; 
	END_IF;
	
	_ManHome.Select := _ManHome.Select AND NOT _ManHome.Interlock;
	IF NOT _ManHome.Select AND NOT _ManHome.Interlock THEN 
		_ManHome.Messages := 'CNC Ready for Selected Axis to be Homed'; 
	END_IF;
	
	_ManHome.Queued := _ManHome.Select;
	IF _ManHome.Queued AND NOT _ManHome.Enabled THEN 
		_ManHome.Messages := 'CNC Waiting for Machine to be put into Resetting'; 
	END_IF;
	
	_ManHome.Enabled := _ManHome.Queued AND Control.PackMLState.Resetting;
	IF _ManHome.Enabled THEN 
		_ManHome.Messages := 'CNC Axis Manual Home Enabled'; 
	END_IF;

//Spindle Warmup
	_SpindleWarmup.Interlock := Spindle.Warm OR (NOT A1_Control.PackMLState.Idle AND NOT A1_Control.PackMLState.Starting AND NOT A1_Control.PackMLState.Execute AND NOT A1_Control.PackMLState.Completing);
	IF _SpindleWarmup.Interlock THEN 
		_SpindleWarmup.Messages := 'Spindle is Warm or CNC is Not in a Suitable State'; 
	END_IF;
	
	_SpindleWarmup.Select := _SpindleWarmup.Select AND NOT _SpindleWarmup.Interlock;
	IF NOT _SpindleWarmup.Select AND NOT _SpindleWarmup.Interlock THEN 
		_SpindleWarmup.Messages := 'Ready for Spindle Warmup'; 
	END_IF;
	
	_SpindleWarmup.Queued := _SpindleWarmup.Select;
	IF _SpindleWarmup.Queued AND NOT _SpindleWarmup.Enabled THEN 
		_SpindleWarmup.Messages := 'Spindle Warmup is Queued'; 
	END_IF;
	
	_SpindleWarmup.Enabled := _SpindleWarmup.Queued AND Control.PackMLState.Execute;
	IF _SpindleWarmup.Enabled THEN 
		_SpindleWarmup.Messages := 'Spindle Warmup Enabled'; 
	END_IF;
	
//Retract Tool
	_RetractTool.Interlock := NOT A1_Control.PackMLState.Idle AND NOT A1_Control.PackMLState.Starting AND NOT A1_Control.PackMLState.Execute AND NOT A1_Control.PackMLState.Completing;
	IF _RetractTool.Interlock THEN 
		_RetractTool.Messages := 'Machine Not in a Suitable State to Retract Tool'; 
	END_IF;
	
	_RetractTool.Select := (_RetractTool.Select) AND NOT _RetractTool.Interlock;
	IF NOT _RetractTool.Select AND NOT _RetractTool.Interlock THEN 
		_RetractTool.Messages := 'Ready for Tool Retract'; 
	END_IF;
	
	_RetractTool.Queued := _RetractTool.Select;
	IF _RetractTool.Queued AND NOT _RetractTool.Enabled THEN 
		_RetractTool.Messages := 'Retract Tool Selection Queued'; 
	END_IF;
	
	_RetractTool.Enabled := _RetractTool.Queued AND Control.PackMLState.Execute;
	IF _RetractTool.Enabled THEN 
		_RetractTool.Messages := 'Retract Tool Enabled'; 
	END_IF;
END_METHOD

METHOD PRIVATE M_Spindle
VAR_INPUT
	{attribute 'tc_no_symbol'}
	_Chan					 : INT;
END_VAR
VAR_INST
	_Delay							: TON;
	_fbHandleSpindleTechno			: HLI3_HandleSpindleTechno;
	_ton							: ARRAY[0..5] OF TON;
	_Step							: UINT;
	_MaxSpeed						: UINT := 24000;
	_r_trig							: ARRAY[0..2] OF R_TRIG;
END_VAR
_fbHandleSpindleTechno(
	nHliAxisIdx:=0, 
	nHliChannelIdx:=_Chan, 	
	bIsChannelSpecific:= TRUE,	
	nRevolution=>Spindle.ComVelocity,
	nLogAxisNoChannelSpecific:= 96, 
	nPosition=> Spindle.Position, 
	bError=> Spindle.Error, 
	nErrorId=> Spindle.ErrorID, 
	M03:= Spindle.M3, 
	M04:= Spindle.M4, 
	M05:= Spindle.M5, 
	M19:= Spindle.M19);

Spindle.ActVelocity:= _Axis[5].stStatus.fActVelo;

// Spindle warm up control
_ton[0](PT:=T#90M, IN:= Spindle.Warm AND NOT SC2501.RunFeedback);
IF _ton[0].Q THEN
	Spindle.Warm := FALSE;
END_IF

CASE _Step OF
	0: //Idle
	IF _SpindleWarmup.Queued THEN
		_Step := 1;
	END_IF
	
	1: //Change to MDI Mode
	_r_trig[0](CLK := TRUE);
	IF _r_trig[0].Q THEN
		_MachineMode[_Chan].MDI := TRUE;
	END_IF

	_MachineMode[_Chan].MDIString := 'T6$R$NM06$R$NM03 S12000$R$NG04 120$R$NM03 S18000$R$NG04 120$R$NM03 S24000$R$NG04 60$R$NM05$R$NT0$R$NM06$R$NG84$R$NM30';
	IF _MachineMode[_Chan].Mode = E_CNC_Mode.MDI_MODE THEN
		_r_trig[0](CLK := FALSE);
		_Step := 2;
		
	ELSIF NOT _SpindleWarmup.Queued THEN
		_Step := 0;
		_MachineMode[_Chan].MDIString := '';
		_MachineMode[_Chan].Standby := TRUE;
	END_IF
	
	2: //Start
	Control.Inputs.Start.Enabled:= TRUE;
	
	IF _MachineMode[_Chan].State = E_CNC_State.ACTIVE AND _SpindleWarmup.Enabled THEN
		_r_trig[0](CLK := FALSE);
		_Step := 3;
	ELSIF NOT _SpindleWarmup.Queued THEN
		_Step := 0;
		_MachineMode[_Chan].MDIString := '';
		_MachineMode[_Chan].Standby := TRUE;
	END_IF
	
	3: //Complete
	IF _ProgramEnd[_Chan] THEN
		Spindle.Warm := TRUE;
		_SpindleWarmup.Select:= FALSE;
		_MachineMode[_Chan].MDIString := '';
		_Step := 0;
		_MachineMode[_Chan].Standby := TRUE;
	ELSIF NOT _SpindleWarmup.Enabled THEN
		_Step := 0;
		_MachineMode[_Chan].MDIString := '';
		_MachineMode[_Chan].Standby := TRUE;
	END_IF
END_CASE
END_METHOD

METHOD PRIVATE M_ToolHandler
VAR_INPUT
	{attribute 'tc_no_symbol'}
	_Chan					 : INT;
END_VAR
VAR_INST
	_r_trig					: ARRAY[0..5] OF R_TRIG;
	_f_trig					: ARRAY[0..2] OF F_TRIG;
	_Step					: UINT;
END_VAR
_ToolData[0].tool_desc.tool_id.basic := 0;
_ToolData[0].tool_desc.valid := TRUE;

//Transfer Tool Data for Requested Tool from Database
IF _Channel[_Chan].pChannel^.ToolData.bToolRequest THEN
	CASE _Channel[_Chan].pChannel^.ToolData.nToolRequestID OF
	0:
		_Channel[_Chan].pChannel^.ToolData.stActTool := _ToolData[0];	
	1:
		_Channel[_Chan].pChannel^.ToolData.stActTool := _ToolData[1];	
	2:
		_Channel[_Chan].pChannel^.ToolData.stActTool := _ToolData[2];	
	3:
		_Channel[_Chan].pChannel^.ToolData.stActTool := _ToolData[3];	
	4:
		_Channel[_Chan].pChannel^.ToolData.stActTool := _ToolData[4];	
	5:
		_Channel[_Chan].pChannel^.ToolData.stActTool := _ToolData[5];	
	6:
		_Channel[_Chan].pChannel^.ToolData.stActTool := _ToolData[6];	
		
	END_CASE		
END_IF

//Transfer Tool Data from Currently used tool back into Database
IF _Channel[_Chan].pChannel^.ToolData.bOldToolDataExist THEN
	_Channel[_Chan].pChannel^.ToolData.bOldToolDataExist := FALSE;
END_IF

//Reply of request read and processed
IF _Channel[_Chan].pChannel^.ToolData.nToolRequestID = _Channel[_Chan].pChannel^.ToolData.stActTool.tool_desc.tool_id.basic THEN
	_Channel[_Chan].pChannel^.ToolData.bToolRequest := FALSE;
END_IF

//Tool Holder
_r_trig[0](CLK:= _Channel[_Chan].pChannel^.M[7].bState_rw);
IF _r_trig[0].Q THEN
	Spindle.M7:= TRUE;
END_IF

_f_trig[0](CLK:= Spindle.M7);
IF _f_trig[0].Q THEN
	_Channel[_Chan].pChannel^.M[7].bState_rw:= FALSE;
END_IF

_r_trig[1](CLK:= _Channel[_Chan].pChannel^.M[8].bState_rw);
IF _r_trig[1].Q THEN
	Spindle.M8:= TRUE;
END_IF

_f_trig[1](CLK:= Spindle.M8);
IF _f_trig[1].Q THEN
	_Channel[_Chan].pChannel^.M[8].bState_rw:= FALSE;
END_IF

_r_trig[2](CLK:= _Channel[_Chan].pChannel^.M[9].bState_rw);
IF _r_trig[2].Q THEN
	Spindle.M9:= TRUE;
END_IF

_f_trig[2](CLK:= Spindle.M9);
IF _f_trig[2].Q THEN
	_Channel[_Chan].pChannel^.M[9].bState_rw:= FALSE;
END_IF

//Tool Retract
IF NOT _RetractTool.Queued THEN
	_Step:= 0;
END_IF

CASE _Step OF
	0: //Idle
	IF _RetractTool.Queued THEN
		_Step := 1;
	END_IF
	
	1: //Change to MDI Mode
	_r_trig[3](CLK := TRUE);
	IF _r_trig[3].Q THEN
		_MachineMode[_Chan].MDI := TRUE;
	END_IF
	
	_MachineMode[_Chan].MDIString := 'G85$R$NX8000 Y650 Z-135 C90 A-90$R$NM02';
	IF _MachineMode[_Chan].Mode = E_CNC_Mode.MDI_MODE THEN
		_r_trig[3](CLK := FALSE);
		_Step := 2;
	END_IF
	
	2: //Start
	Control.Inputs.Start.Select:= TRUE;
	
	IF _MachineMode[_Chan].State = E_CNC_State.ACTIVE THEN
		_Step := 3;
	END_IF
	
	3: //Complete
	IF _ProgramEnd[_Chan] THEN//_MachineMode[_Chan].State = E_CNC_State.READY THEN
		_Step := 0;
		_MachineMode[_Chan].MDIString := '';
		_RetractTool.Select:= FALSE;
		_MachineMode[_Chan].Standby := TRUE;
	END_IF
END_CASE
END_METHOD

METHOD PRIVATE M_VariableViewer
VAR_INST
	_fbReadCNCVariables 	: FB_ReadCNCVariables;
END_VAR
_fbReadCNCVariables(
	bEnable:= TRUE, 
	nChanIdx:= _SelectedChannel, 
	eVariablesType:= eVariablesType, 
	tIntervall:= T#1S, 	 
	stCNCVariablesViewer_Data:= stCNCVariablesViewer_Data);

_pVE_Chan0:= HLI3_LinkVEChannelStructure(nChanIdx:= 0, bGlobal:= FALSE);

_pVE_Chan0^.ParkPos.X:=  _ParkPositions[0];
_pVE_Chan0^.ParkPos.Y:=  _ParkPositions[1];
_pVE_Chan0^.ParkPos.Z:=  _ParkPositions[2];
_pVE_Chan0^.ParkPos.C:=  _ParkPositions[3];
_pVE_Chan0^.ParkPos.A:=  _ParkPositions[4];
END_METHOD

METHOD PRIVATE M_WarningMonitor
VAR_INPUT
END_VAR
VAR_INST
END_VAR
VAR_INST // added by the converter: edge detectors and wires of the graphical bodies
    _w1 : BOOL;
END_VAR
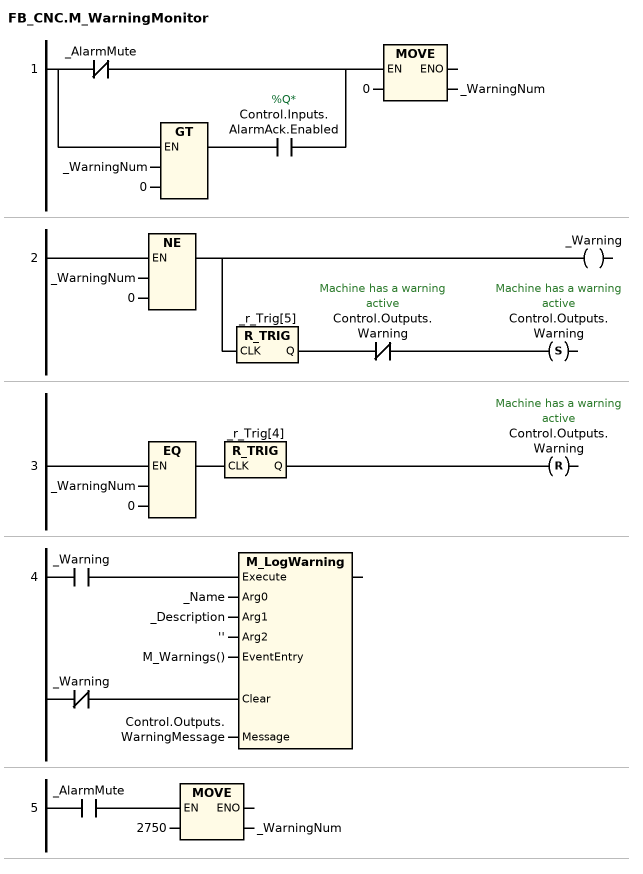
// NETWORK 1
//   Control.Inputs.AlarmAck.Enabled: AT %Q*
IF NOT _AlarmMute OR _WarningNum > 0 AND Control.Inputs.AlarmAck.Enabled THEN _WarningNum := 0; END_IF

// NETWORK 2
//   Control.Outputs.Warning: Machine has a warning active
_w1 := _WarningNum <> 0;
_Warning := _w1;
_r_Trig[5](CLK := _w1); // R_TRIG
Control.Outputs.Warning S= _r_Trig[5].Q AND NOT Control.Outputs.Warning;

// NETWORK 3
//   Control.Outputs.Warning: Machine has a warning active
_r_Trig[4](CLK := _WarningNum = 0); // R_TRIG
Control.Outputs.Warning R= _r_Trig[4].Q;

// NETWORK 4
M_LogWarning(Execute := _Warning, Arg0 := _Name, Arg1 := _Description, Arg2 := '', EventEntry := M_Warnings(), Clear := NOT _Warning, Message := Control.Outputs.WarningMessage);

// NETWORK 5
IF _AlarmMute THEN _WarningNum := 2750; END_IF
END_METHOD

METHOD PRIVATE M_Warnings : TcEventEntry
VAR_INPUT
END_VAR
CASE _WarningNum OF		
	2750: M_Warnings:= TC_Events.TcCnc.W_2750;//Alarm Mute Active						
ELSE
	M_Warnings:=  TC_Events.TcCnc.W_Undefined;
END_CASE
END_METHOD

PROPERTY PUBLIC MachineMode : REFERENCE TO ARRAY[0..3] OF ST_MachineMode;
GET
MachineMode REF= _MachineMode;
END_GET
END_PROPERTY

{attribute 'monitoring' := 'variable'}
PROPERTY PUBLIC Name : String[15]
GET
Name := _Name;
END_GET
SET
_Name := Name;
END_SET
END_PROPERTY

PROPERTY PUBLIC ProgramEnd : REFERENCE TO ARRAY[0..3] OF  BOOL
GET
ProgramEnd REF= _ProgramEnd;
END_GET
END_PROPERTY

PROPERTY PUBLIC ToolData : ARRAY [0..6] OF ST_CNC_TOOL_DATA_EXT
SET
_ToolData:= ToolData;
END_SET
END_PROPERTY

PROPERTY PUBLIC Variables : REFERENCE TO ARRAY[0..9] OF ST_Variable
GET
Variables REF= _Variables;
END_GET
END_PROPERTY

{attribute 'monitoring' := 'variable'}
PROPERTY PUBLIC Warning : Bool
GET
Warning := _Warning;
END_GET
END_PROPERTY

END_FUNCTION_BLOCK

(* stored: Version 1.1.0.1, ProductVersion 3.1.4024.3
   POU FB_CNC: Id {cf2e5201-7a65-4bdf-9557-5bc64b9a3b2c}, SpecialFunc None
   Property Alarm: Id {359f4eee-d9a0-4521-962e-f7d57982a541}
   Get Get: Id {61388294-419b-458f-bc2b-b3e2226a6579}
   Property AlarmMute: Id {7948eba6-0c41-4756-9ef3-f982bead2b79}
   Set Set: Id {963ade74-b216-469b-afc1-68758f2cec2e}
   Property AutoHome: Id {ab395135-4b23-4f9a-a0dd-ccd5102cd195}
   Set Set: Id {7b5c1eb4-837a-48b9-9b69-465a72284bb5}
   Property AxisEnabled: Id {69ff1fbf-98be-452d-ae1a-78bb861e8efd}
   Get Get: Id {7d84d92b-d133-42b4-a75f-ff425b45cf44}
   Property Description: Id {40aa6561-11c0-4b28-872b-7fb5653ac56e}
   Get Get: Id {05ef46eb-f8a5-4005-8766-e7700868af57}
   Set Set: Id {1d7ebb25-99e6-4c7e-885b-8d44a9870fa9}
   Property Fault: Id {fb7aa23f-5e73-4c0d-be57-4d847db5941c}
   Set Set: Id {1894d889-4160-4322-aa06-e59987e132df}
   Property FaultTimer_ET: Id {7e22a7dd-22a3-4dd1-ab54-9897ee6bb3a0}
   Get Get: Id {d4c923a8-596e-4647-82f8-21dfd92d7684}
   Property FaultTimer_PT: Id {824f0c37-26db-4081-a4ee-f0548ace22e9}
   Get Get: Id {c7a44f53-7cef-4367-b3f8-3ba50b57c69c}
   Set Set: Id {644aedff-272b-4e1d-8d0a-b6788272f907}
   Property FeedOverride: Id {80a7a54e-5404-4a02-9c83-808a38edf8bc}
   Get Get: Id {18ff8965-7c22-4954-8a19-06eea85069db}
   Set Set: Id {dfae57c9-a52b-4b29-b621-d516d84695c1}
   Property HandwheelSelected: Id {eab7aa11-8243-44da-b78b-103a0ea97542}
   Get Get: Id {33c9364a-ad92-4848-8838-97915c2fed3d}
   Property Homed: Id {0ba18c2e-6a1b-4a41-8c0b-6818ced9f199}
   Get Get: Id {3447c266-c031-4c0f-a7e6-f1292d29f1ee}
   Method M_AlarmMonitor: Id {551bc7b8-11df-43f3-9985-4613b8af0d4d}
   Method M_Alarms: Id {ff3115cc-2cf8-4aba-b81e-75da85fbc3bf}
   Method M_AxesHandler: Id {93ad86df-0a10-4356-bf08-23fe58533ff5}
   Method M_ChannelHandler: Id {0a8dacf7-3655-49c6-a433-af25632fc464}
   Method M_Homing: Id {466dc8fd-1909-44dc-af82-e5fad6e99017}
   Method M_ManualMode: Id {6c94a58e-1d14-4232-9b46-07e75cdeb92e}
   Method M_Selections: Id {be37a95d-35cb-48bf-bcf9-2fb9ab9d4d86}
   Method M_Spindle: Id {e64b7526-e6ce-49bf-bddc-c74afdc22bd2}
   Method M_ToolHandler: Id {9e892e2a-8d72-42cc-89f7-4f9f6b768fcd}
   Method M_VariableViewer: Id {2919cdc1-60b3-44aa-9241-4a23b53a6fe0}
   Method M_WarningMonitor: Id {dd29c373-e592-4892-8644-e81c2f8ce1e5}
   Method M_Warnings: Id {1f82e3c5-6c32-4405-b4b7-c1a6ab9217ef}
   Property MachineMode: Id {35200c78-ca0f-4c0a-a146-c4e657d8f6b9}
   Get Get: Id {44f7035f-e36e-4c08-84fa-d4979fd47328}
   Property Name: Id {6bcb0b1f-af97-4ff4-a4ad-20fe9a6bd558}
   Get Get: Id {a6201308-7280-4eb8-b725-8437625eded9}
   Set Set: Id {46e93fdb-d817-4dc2-aa27-428824e675c2}
   Property ProgramEnd: Id {751a4dba-0a63-4a74-a46d-bba737826f15}
   Get Get: Id {e07d12d1-46ff-42e3-a141-16df3f15f53b}
   Property ToolData: Id {a1ed01ca-de70-408b-b241-baa0bbe38e00}
   Set Set: Id {bc730669-cd4c-40db-81cd-d3901e8c0c32}
   Property Variables: Id {54cae200-5400-473e-8e73-34ec6e4a47c2}
   Get Get: Id {f126b3d3-ae41-4df2-9ed7-26eb92202520}
   Property Warning: Id {7520702d-73cd-4668-96a8-1f71043a3dec}
   Get Get: Id {dc54e4cc-a070-4a07-a294-b673225a685a} *)
